(* :Description:  This function is used to convert string into bytes structure, ready to send it via TCP/IP protocole *)
FUNCTION FUN_StringToTcpBufferData : BOOL
VAR_INPUT
	sMessageAddr 	: PVOID;					(* Source string message *)
	stSendDataAddr	: PVOID;					(* Destination TCP/IP data structure *)
END_VAR
VAR
	psMessage	: POINTER TO STRING;			(* Pointer to string converted to structure *)
	pstSendData	: POINTER TO ST_TcpBufferData;	(* Pointer to structure made of string bytes *)
END_VAR

(* Check if any input address is different than zero*)
IF sMessageAddr <> 0 AND stSendDataAddr <> 0 THEN
	(* Access to adress*)
	psMessage := sMessageAddr;
	pstSendData := stSendDataAddr;
	
	pstSendData^.iLength := INT_TO_UDINT(LEN(psMessage^));
	
	(* Copy bytes from string to structure *)
	MEMCPY(destAddr := stSendDataAddr, srcAddr := sMessageAddr, n := pstSendData^.iLength);

	(* Function done *)
	FUN_StringToTcpBufferData := TRUE;
(* One of adresses was not correct *)
ELSE
	FUN_StringToTcpBufferData := FALSE;
END_IF

END_FUNCTION

(* stored: Version 1.1.0.1, ProductVersion 3.1.4024.12
   POU FUN_StringToTcpBufferData: Id {634c64f8-7380-48ba-ba53-78cc0223e1e3}, SpecialFunc None *)
